FUNCTION_BLOCK FB_Properties

PROPERTY Count : INT
GET
END_GET
END_PROPERTY

PROPERTY Name : STRING
GET
END_GET
SET
END_SET
END_PROPERTY

END_FUNCTION_BLOCK

(* stored: Version 1.1.0.1
   POU FB_Properties: Id {11111111-1111-1111-1111-111111111104}
   Property Count: Id {33333333-3333-3333-3333-333333333301}
   Get Get: Id {33333333-3333-3333-3333-333333333302}
   Property Name: Id {33333333-3333-3333-3333-333333333303}
   Get Get: Id {33333333-3333-3333-3333-333333333304}
   Set Set: Id {33333333-3333-3333-3333-333333333305} *)
